// TIA Portal V16 export
// export: Created 2023-03-29T11:04:41.0167159Z, ExportSetting WithDefaults, DisplayName Totally Integrated Automation Portal, DisplayVersion V16 Update 6, DisplayName TIA Portal Version Control Interface, DisplayVersion V16 Update 2, DisplayName TIA Portal Openness, DisplayVersion V16 Update 6, DisplayName STEP 7 Professional, DisplayVersion V16 Update 6, DisplayName STEP 7 Safety, DisplayVersion V16, DisplayName WinCC Advanced, DisplayVersion V16 Update 6
FUNCTION "Synchroniczna_wymiana_danych_PLC1-PLC2" : Void   // FC61, LAD
TITLE = Wymiana danych
{ S7_Optimized_Access := 'TRUE' }
AUTHOR : rtecmer
VERSION : 0.1
// Funkcja grupuje bloki funkcji służąc wymianie danych HMI - PLC1, HMI-PLC2 i SCADA. Wprowadzanie wartości z poziomu HMI Zbiorniki lub HMI Pompownia czy SCADA jest nadpisywane w docelowym sterowniku. Zmian włónych parametrów układu sterowania pompownią, zbiornikami można dokonywać w dowolnego miejsca.
// stored: AutoNumber true, IsIECCheckEnabled false, SetENOAutomatically false, UDAEnableTagReadback false
   VAR_TEMP   // added for the SCL form of the ladder/FBD networks
      _w1 : Bool;
   END_VAR
BEGIN

REGION Network 2: Detekcja zmiany danych - Poziom napełnienia
   // Wymiana danych między PLC 1, PLC 2, SCADA
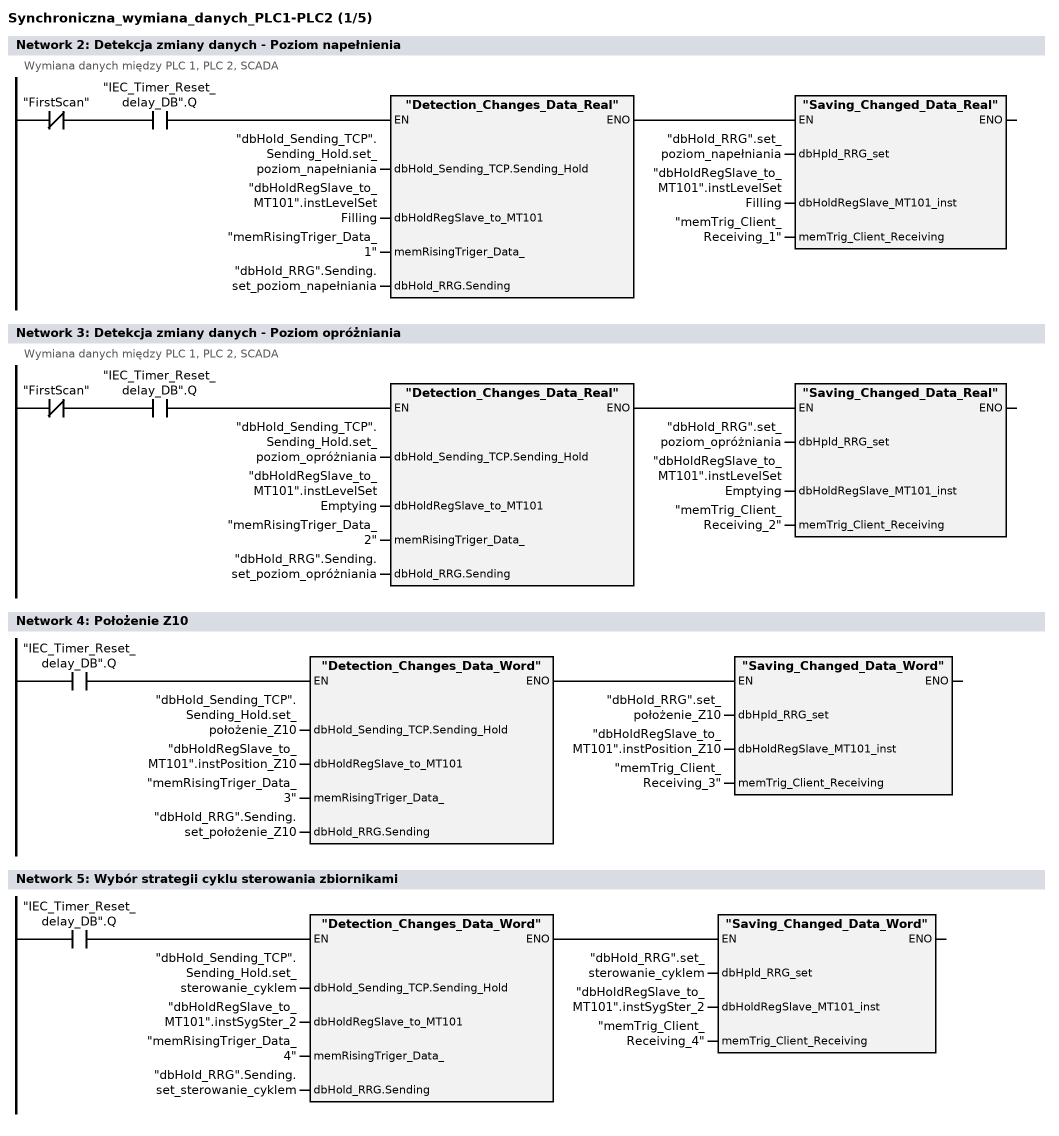
   RUNG wire#powerrail
      I_Contact( "FirstScan" )
      Contact( "IEC_Timer_Reset_delay_DB".Q )
      "Detection_Changes_Data_Real"("dbHold_Sending_TCP.Sending_Hold" := "dbHold_Sending_TCP".Sending_Hold.set_poziom_napełniania, dbHoldRegSlave_to_MT101 := "dbHoldRegSlave_to_MT101".instLevelSetFilling, memRisingTriger_Data_ := "memRisingTriger_Data_1", "dbHold_RRG.Sending" := "dbHold_RRG".Sending.set_poziom_napełniania)
      "Saving_Changed_Data_Real"(dbHpld_RRG_set := "dbHold_RRG".set_poziom_napełniania, dbHoldRegSlave_MT101_inst := "dbHoldRegSlave_to_MT101".instLevelSetFilling, memTrig_Client_Receiving := "memTrig_Client_Receiving_1")
   END_RUNG
   // the same network as SCL:
   "Detection_Changes_Data_Real"(EN := NOT "FirstScan" AND "IEC_Timer_Reset_delay_DB".Q,
                           "dbHold_Sending_TCP.Sending_Hold" := "dbHold_Sending_TCP".Sending_Hold.set_poziom_napełniania,
                           dbHoldRegSlave_to_MT101 := "dbHoldRegSlave_to_MT101".instLevelSetFilling,
                           memRisingTriger_Data_ := "memRisingTriger_Data_1",
                           "dbHold_RRG.Sending" := "dbHold_RRG".Sending.set_poziom_napełniania,
                           ENO => #_w1);
   IF #_w1 THEN
       "Saving_Changed_Data_Real"(dbHpld_RRG_set := "dbHold_RRG".set_poziom_napełniania,
                               dbHoldRegSlave_MT101_inst := "dbHoldRegSlave_to_MT101".instLevelSetFilling,
                               memTrig_Client_Receiving := "memTrig_Client_Receiving_1");
   END_IF;
END_REGION

REGION Network 3: Detekcja zmiany danych - Poziom opróżniania
   // Wymiana danych między PLC 1, PLC 2, SCADA
   RUNG wire#powerrail
      I_Contact( "FirstScan" )
      Contact( "IEC_Timer_Reset_delay_DB".Q )
      "Detection_Changes_Data_Real"("dbHold_Sending_TCP.Sending_Hold" := "dbHold_Sending_TCP".Sending_Hold.set_poziom_opróżniania, dbHoldRegSlave_to_MT101 := "dbHoldRegSlave_to_MT101".instLevelSetEmptying, memRisingTriger_Data_ := "memRisingTriger_Data_2", "dbHold_RRG.Sending" := "dbHold_RRG".Sending.set_poziom_opróżniania)
      "Saving_Changed_Data_Real"(dbHpld_RRG_set := "dbHold_RRG".set_poziom_opróżniania, dbHoldRegSlave_MT101_inst := "dbHoldRegSlave_to_MT101".instLevelSetEmptying, memTrig_Client_Receiving := "memTrig_Client_Receiving_2")
   END_RUNG
   // the same network as SCL:
   "Detection_Changes_Data_Real"(EN := NOT "FirstScan" AND "IEC_Timer_Reset_delay_DB".Q,
                           "dbHold_Sending_TCP.Sending_Hold" := "dbHold_Sending_TCP".Sending_Hold.set_poziom_opróżniania,
                           dbHoldRegSlave_to_MT101 := "dbHoldRegSlave_to_MT101".instLevelSetEmptying,
                           memRisingTriger_Data_ := "memRisingTriger_Data_2",
                           "dbHold_RRG.Sending" := "dbHold_RRG".Sending.set_poziom_opróżniania,
                           ENO => #_w1);
   IF #_w1 THEN
       "Saving_Changed_Data_Real"(dbHpld_RRG_set := "dbHold_RRG".set_poziom_opróżniania,
                               dbHoldRegSlave_MT101_inst := "dbHoldRegSlave_to_MT101".instLevelSetEmptying,
                               memTrig_Client_Receiving := "memTrig_Client_Receiving_2");
   END_IF;
END_REGION

REGION Network 4: Położenie Z10
   RUNG wire#powerrail
      Contact( "IEC_Timer_Reset_delay_DB".Q )
      "Detection_Changes_Data_Word"("dbHold_Sending_TCP.Sending_Hold" := "dbHold_Sending_TCP".Sending_Hold.set_położenie_Z10, dbHoldRegSlave_to_MT101 := "dbHoldRegSlave_to_MT101".instPosition_Z10, memRisingTriger_Data_ := "memRisingTriger_Data_3", "dbHold_RRG.Sending" := "dbHold_RRG".Sending.set_położenie_Z10)
      "Saving_Changed_Data_Word"(dbHpld_RRG_set := "dbHold_RRG".set_położenie_Z10, dbHoldRegSlave_MT101_inst := "dbHoldRegSlave_to_MT101".instPosition_Z10, memTrig_Client_Receiving := "memTrig_Client_Receiving_3")
   END_RUNG
   // the same network as SCL:
   "Detection_Changes_Data_Word"(EN := "IEC_Timer_Reset_delay_DB".Q,
                           "dbHold_Sending_TCP.Sending_Hold" := "dbHold_Sending_TCP".Sending_Hold.set_położenie_Z10,
                           dbHoldRegSlave_to_MT101 := "dbHoldRegSlave_to_MT101".instPosition_Z10,
                           memRisingTriger_Data_ := "memRisingTriger_Data_3",
                           "dbHold_RRG.Sending" := "dbHold_RRG".Sending.set_położenie_Z10,
                           ENO => #_w1);
   IF #_w1 THEN
       "Saving_Changed_Data_Word"(dbHpld_RRG_set := "dbHold_RRG".set_położenie_Z10,
                               dbHoldRegSlave_MT101_inst := "dbHoldRegSlave_to_MT101".instPosition_Z10,
                               memTrig_Client_Receiving := "memTrig_Client_Receiving_3");
   END_IF;
END_REGION

REGION Network 5: Wybór strategii cyklu sterowania zbiornikami
   RUNG wire#powerrail
      Contact( "IEC_Timer_Reset_delay_DB".Q )
      "Detection_Changes_Data_Word"("dbHold_Sending_TCP.Sending_Hold" := "dbHold_Sending_TCP".Sending_Hold.set_sterowanie_cyklem, dbHoldRegSlave_to_MT101 := "dbHoldRegSlave_to_MT101".instSygSter_2, memRisingTriger_Data_ := "memRisingTriger_Data_4", "dbHold_RRG.Sending" := "dbHold_RRG".Sending.set_sterowanie_cyklem)
      "Saving_Changed_Data_Word"(dbHpld_RRG_set := "dbHold_RRG".set_sterowanie_cyklem, dbHoldRegSlave_MT101_inst := "dbHoldRegSlave_to_MT101".instSygSter_2, memTrig_Client_Receiving := "memTrig_Client_Receiving_4")
   END_RUNG
   // the same network as SCL:
   "Detection_Changes_Data_Word"(EN := "IEC_Timer_Reset_delay_DB".Q,
                           "dbHold_Sending_TCP.Sending_Hold" := "dbHold_Sending_TCP".Sending_Hold.set_sterowanie_cyklem,
                           dbHoldRegSlave_to_MT101 := "dbHoldRegSlave_to_MT101".instSygSter_2,
                           memRisingTriger_Data_ := "memRisingTriger_Data_4",
                           "dbHold_RRG.Sending" := "dbHold_RRG".Sending.set_sterowanie_cyklem,
                           ENO => #_w1);
   IF #_w1 THEN
       "Saving_Changed_Data_Word"(dbHpld_RRG_set := "dbHold_RRG".set_sterowanie_cyklem,
                               dbHoldRegSlave_MT101_inst := "dbHoldRegSlave_to_MT101".instSygSter_2,
                               memTrig_Client_Receiving := "memTrig_Client_Receiving_4");
   END_IF;
END_REGION

REGION Network 6: Godzina napełniania start
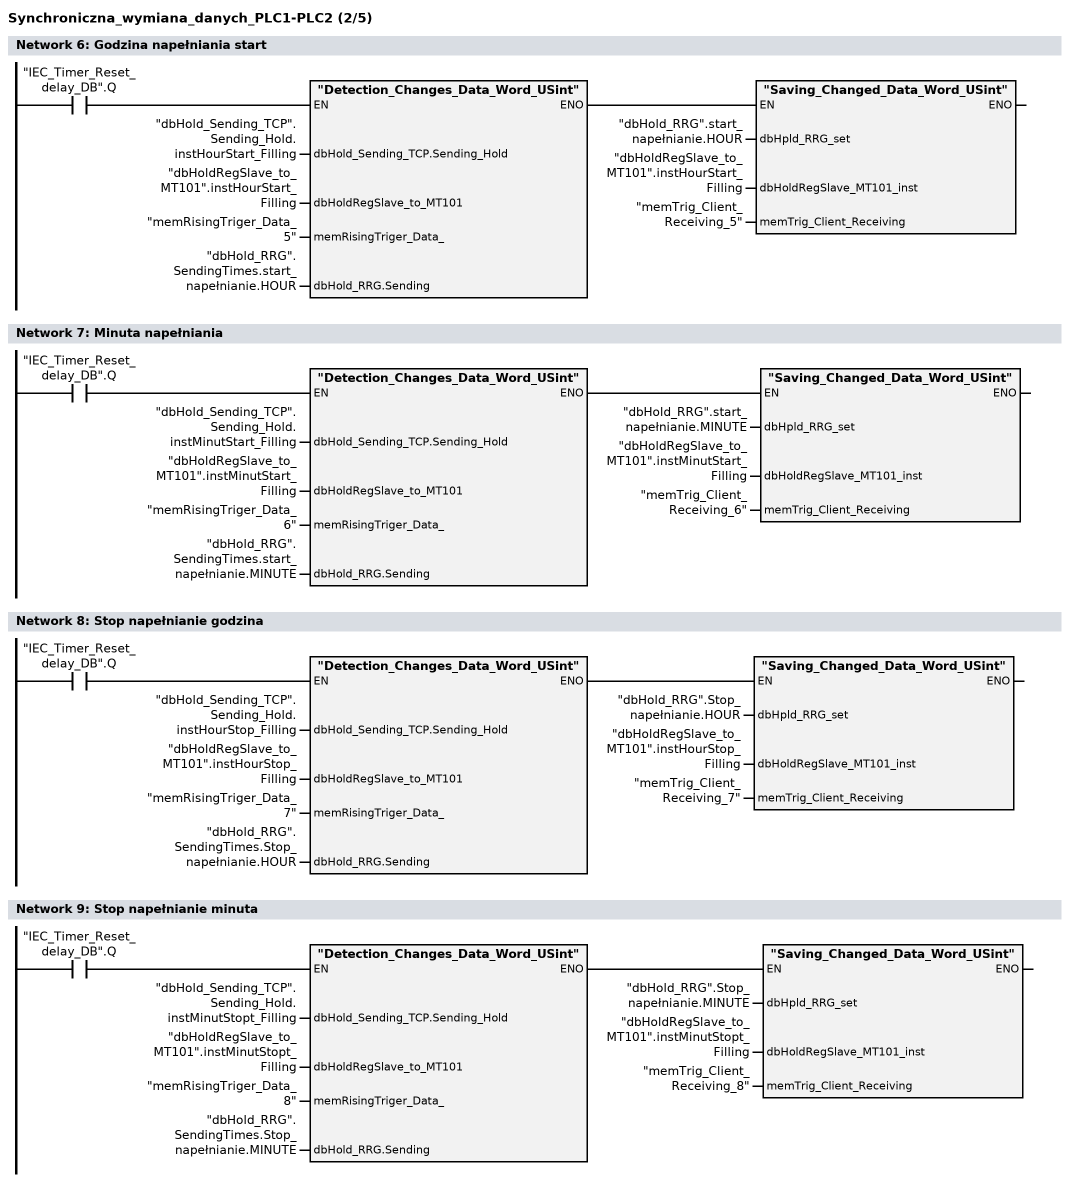
   RUNG wire#powerrail
      Contact( "IEC_Timer_Reset_delay_DB".Q )
      "Detection_Changes_Data_Word_USint"("dbHold_Sending_TCP.Sending_Hold" := "dbHold_Sending_TCP".Sending_Hold.instHourStart_Filling, dbHoldRegSlave_to_MT101 := "dbHoldRegSlave_to_MT101".instHourStart_Filling, memRisingTriger_Data_ := "memRisingTriger_Data_5", "dbHold_RRG.Sending" := "dbHold_RRG".SendingTimes.start_napełnianie.HOUR)
      "Saving_Changed_Data_Word_USint"(dbHpld_RRG_set := "dbHold_RRG".start_napełnianie.HOUR, dbHoldRegSlave_MT101_inst := "dbHoldRegSlave_to_MT101".instHourStart_Filling, memTrig_Client_Receiving := "memTrig_Client_Receiving_5")
   END_RUNG
   // the same network as SCL:
   "Detection_Changes_Data_Word_USint"(EN := "IEC_Timer_Reset_delay_DB".Q,
                           "dbHold_Sending_TCP.Sending_Hold" := "dbHold_Sending_TCP".Sending_Hold.instHourStart_Filling,
                           dbHoldRegSlave_to_MT101 := "dbHoldRegSlave_to_MT101".instHourStart_Filling,
                           memRisingTriger_Data_ := "memRisingTriger_Data_5",
                           "dbHold_RRG.Sending" := "dbHold_RRG".SendingTimes.start_napełnianie.HOUR,
                           ENO => #_w1);
   IF #_w1 THEN
       "Saving_Changed_Data_Word_USint"(dbHpld_RRG_set := "dbHold_RRG".start_napełnianie.HOUR,
                               dbHoldRegSlave_MT101_inst := "dbHoldRegSlave_to_MT101".instHourStart_Filling,
                               memTrig_Client_Receiving := "memTrig_Client_Receiving_5");
   END_IF;
END_REGION

REGION Network 7: Minuta napełniania
   RUNG wire#powerrail
      Contact( "IEC_Timer_Reset_delay_DB".Q )
      "Detection_Changes_Data_Word_USint"("dbHold_Sending_TCP.Sending_Hold" := "dbHold_Sending_TCP".Sending_Hold.instMinutStart_Filling, dbHoldRegSlave_to_MT101 := "dbHoldRegSlave_to_MT101".instMinutStart_Filling, memRisingTriger_Data_ := "memRisingTriger_Data_6", "dbHold_RRG.Sending" := "dbHold_RRG".SendingTimes.start_napełnianie.MINUTE)
      "Saving_Changed_Data_Word_USint"(dbHpld_RRG_set := "dbHold_RRG".start_napełnianie.MINUTE, dbHoldRegSlave_MT101_inst := "dbHoldRegSlave_to_MT101".instMinutStart_Filling, memTrig_Client_Receiving := "memTrig_Client_Receiving_6")
   END_RUNG
   // the same network as SCL:
   "Detection_Changes_Data_Word_USint"(EN := "IEC_Timer_Reset_delay_DB".Q,
                           "dbHold_Sending_TCP.Sending_Hold" := "dbHold_Sending_TCP".Sending_Hold.instMinutStart_Filling,
                           dbHoldRegSlave_to_MT101 := "dbHoldRegSlave_to_MT101".instMinutStart_Filling,
                           memRisingTriger_Data_ := "memRisingTriger_Data_6",
                           "dbHold_RRG.Sending" := "dbHold_RRG".SendingTimes.start_napełnianie.MINUTE,
                           ENO => #_w1);
   IF #_w1 THEN
       "Saving_Changed_Data_Word_USint"(dbHpld_RRG_set := "dbHold_RRG".start_napełnianie.MINUTE,
                               dbHoldRegSlave_MT101_inst := "dbHoldRegSlave_to_MT101".instMinutStart_Filling,
                               memTrig_Client_Receiving := "memTrig_Client_Receiving_6");
   END_IF;
END_REGION

REGION Network 8: Stop napełnianie godzina
   RUNG wire#powerrail
      Contact( "IEC_Timer_Reset_delay_DB".Q )
      "Detection_Changes_Data_Word_USint"("dbHold_Sending_TCP.Sending_Hold" := "dbHold_Sending_TCP".Sending_Hold.instHourStop_Filling, dbHoldRegSlave_to_MT101 := "dbHoldRegSlave_to_MT101".instHourStop_Filling, memRisingTriger_Data_ := "memRisingTriger_Data_7", "dbHold_RRG.Sending" := "dbHold_RRG".SendingTimes.Stop_napełnianie.HOUR)
      "Saving_Changed_Data_Word_USint"(dbHpld_RRG_set := "dbHold_RRG".Stop_napełnianie.HOUR, dbHoldRegSlave_MT101_inst := "dbHoldRegSlave_to_MT101".instHourStop_Filling, memTrig_Client_Receiving := "memTrig_Client_Receiving_7")
   END_RUNG
   // the same network as SCL:
   "Detection_Changes_Data_Word_USint"(EN := "IEC_Timer_Reset_delay_DB".Q,
                           "dbHold_Sending_TCP.Sending_Hold" := "dbHold_Sending_TCP".Sending_Hold.instHourStop_Filling,
                           dbHoldRegSlave_to_MT101 := "dbHoldRegSlave_to_MT101".instHourStop_Filling,
                           memRisingTriger_Data_ := "memRisingTriger_Data_7",
                           "dbHold_RRG.Sending" := "dbHold_RRG".SendingTimes.Stop_napełnianie.HOUR,
                           ENO => #_w1);
   IF #_w1 THEN
       "Saving_Changed_Data_Word_USint"(dbHpld_RRG_set := "dbHold_RRG".Stop_napełnianie.HOUR,
                               dbHoldRegSlave_MT101_inst := "dbHoldRegSlave_to_MT101".instHourStop_Filling,
                               memTrig_Client_Receiving := "memTrig_Client_Receiving_7");
   END_IF;
END_REGION

REGION Network 9: Stop napełnianie minuta
   RUNG wire#powerrail
      Contact( "IEC_Timer_Reset_delay_DB".Q )
      "Detection_Changes_Data_Word_USint"("dbHold_Sending_TCP.Sending_Hold" := "dbHold_Sending_TCP".Sending_Hold.instMinutStopt_Filling, dbHoldRegSlave_to_MT101 := "dbHoldRegSlave_to_MT101".instMinutStopt_Filling, memRisingTriger_Data_ := "memRisingTriger_Data_8", "dbHold_RRG.Sending" := "dbHold_RRG".SendingTimes.Stop_napełnianie.MINUTE)
      "Saving_Changed_Data_Word_USint"(dbHpld_RRG_set := "dbHold_RRG".Stop_napełnianie.MINUTE, dbHoldRegSlave_MT101_inst := "dbHoldRegSlave_to_MT101".instMinutStopt_Filling, memTrig_Client_Receiving := "memTrig_Client_Receiving_8")
   END_RUNG
   // the same network as SCL:
   "Detection_Changes_Data_Word_USint"(EN := "IEC_Timer_Reset_delay_DB".Q,
                           "dbHold_Sending_TCP.Sending_Hold" := "dbHold_Sending_TCP".Sending_Hold.instMinutStopt_Filling,
                           dbHoldRegSlave_to_MT101 := "dbHoldRegSlave_to_MT101".instMinutStopt_Filling,
                           memRisingTriger_Data_ := "memRisingTriger_Data_8",
                           "dbHold_RRG.Sending" := "dbHold_RRG".SendingTimes.Stop_napełnianie.MINUTE,
                           ENO => #_w1);
   IF #_w1 THEN
       "Saving_Changed_Data_Word_USint"(dbHpld_RRG_set := "dbHold_RRG".Stop_napełnianie.MINUTE,
                               dbHoldRegSlave_MT101_inst := "dbHoldRegSlave_to_MT101".instMinutStopt_Filling,
                               memTrig_Client_Receiving := "memTrig_Client_Receiving_8");
   END_IF;
END_REGION

REGION Network 10: Start przetłaczanie (miasto) godzina
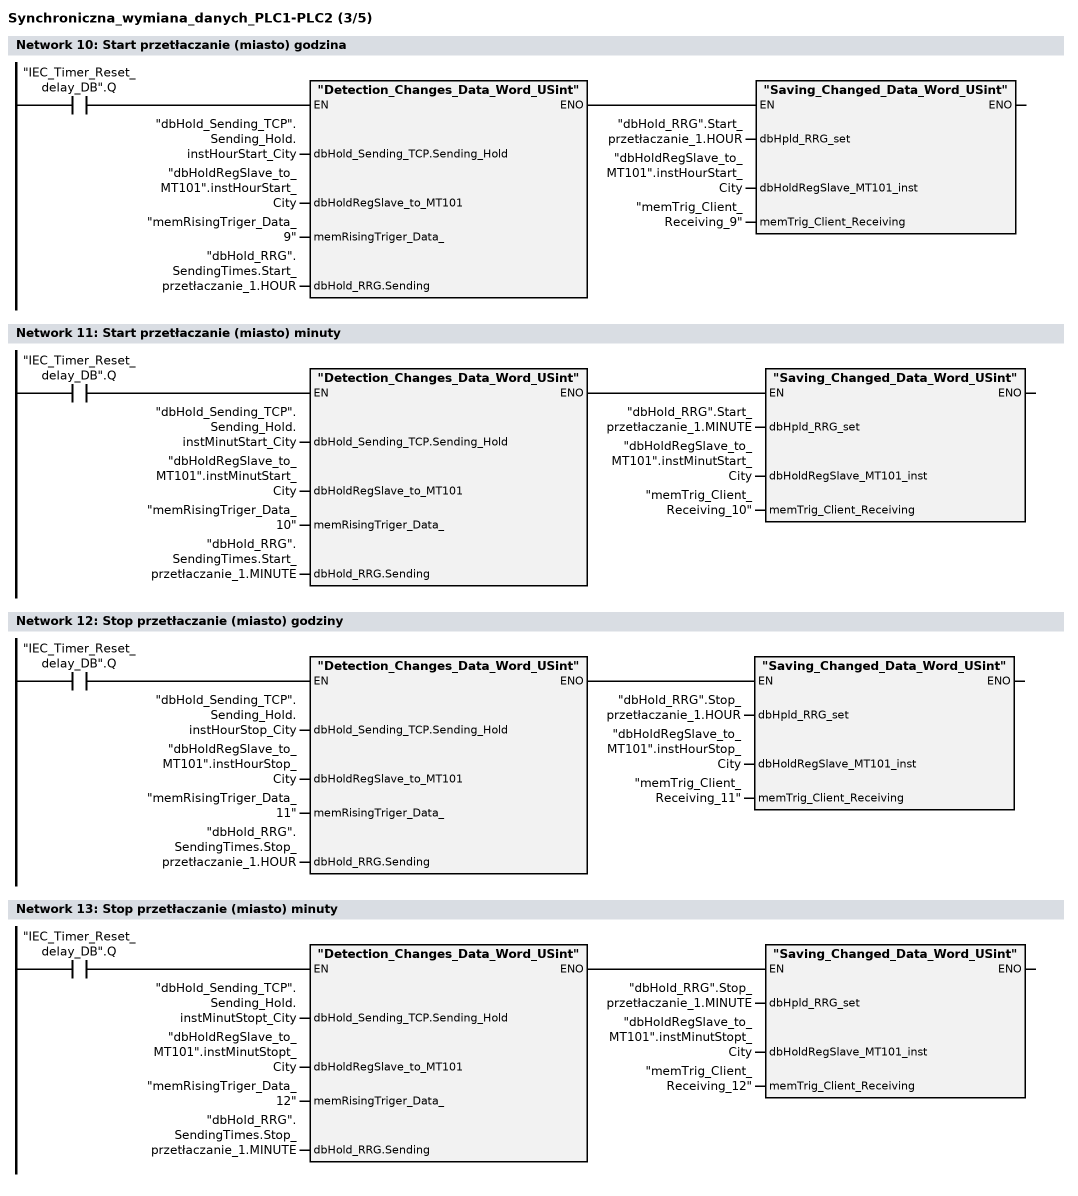
   RUNG wire#powerrail
      Contact( "IEC_Timer_Reset_delay_DB".Q )
      "Detection_Changes_Data_Word_USint"("dbHold_Sending_TCP.Sending_Hold" := "dbHold_Sending_TCP".Sending_Hold.instHourStart_City, dbHoldRegSlave_to_MT101 := "dbHoldRegSlave_to_MT101".instHourStart_City, memRisingTriger_Data_ := "memRisingTriger_Data_9", "dbHold_RRG.Sending" := "dbHold_RRG".SendingTimes.Start_przetłaczanie_1.HOUR)
      "Saving_Changed_Data_Word_USint"(dbHpld_RRG_set := "dbHold_RRG".Start_przetłaczanie_1.HOUR, dbHoldRegSlave_MT101_inst := "dbHoldRegSlave_to_MT101".instHourStart_City, memTrig_Client_Receiving := "memTrig_Client_Receiving_9")
   END_RUNG
   // the same network as SCL:
   "Detection_Changes_Data_Word_USint"(EN := "IEC_Timer_Reset_delay_DB".Q,
                           "dbHold_Sending_TCP.Sending_Hold" := "dbHold_Sending_TCP".Sending_Hold.instHourStart_City,
                           dbHoldRegSlave_to_MT101 := "dbHoldRegSlave_to_MT101".instHourStart_City,
                           memRisingTriger_Data_ := "memRisingTriger_Data_9",
                           "dbHold_RRG.Sending" := "dbHold_RRG".SendingTimes.Start_przetłaczanie_1.HOUR,
                           ENO => #_w1);
   IF #_w1 THEN
       "Saving_Changed_Data_Word_USint"(dbHpld_RRG_set := "dbHold_RRG".Start_przetłaczanie_1.HOUR,
                               dbHoldRegSlave_MT101_inst := "dbHoldRegSlave_to_MT101".instHourStart_City,
                               memTrig_Client_Receiving := "memTrig_Client_Receiving_9");
   END_IF;
END_REGION

REGION Network 11: Start przetłaczanie (miasto) minuty
   RUNG wire#powerrail
      Contact( "IEC_Timer_Reset_delay_DB".Q )
      "Detection_Changes_Data_Word_USint"("dbHold_Sending_TCP.Sending_Hold" := "dbHold_Sending_TCP".Sending_Hold.instMinutStart_City, dbHoldRegSlave_to_MT101 := "dbHoldRegSlave_to_MT101".instMinutStart_City, memRisingTriger_Data_ := "memRisingTriger_Data_10", "dbHold_RRG.Sending" := "dbHold_RRG".SendingTimes.Start_przetłaczanie_1.MINUTE)
      "Saving_Changed_Data_Word_USint"(dbHpld_RRG_set := "dbHold_RRG".Start_przetłaczanie_1.MINUTE, dbHoldRegSlave_MT101_inst := "dbHoldRegSlave_to_MT101".instMinutStart_City, memTrig_Client_Receiving := "memTrig_Client_Receiving_10")
   END_RUNG
   // the same network as SCL:
   "Detection_Changes_Data_Word_USint"(EN := "IEC_Timer_Reset_delay_DB".Q,
                           "dbHold_Sending_TCP.Sending_Hold" := "dbHold_Sending_TCP".Sending_Hold.instMinutStart_City,
                           dbHoldRegSlave_to_MT101 := "dbHoldRegSlave_to_MT101".instMinutStart_City,
                           memRisingTriger_Data_ := "memRisingTriger_Data_10",
                           "dbHold_RRG.Sending" := "dbHold_RRG".SendingTimes.Start_przetłaczanie_1.MINUTE,
                           ENO => #_w1);
   IF #_w1 THEN
       "Saving_Changed_Data_Word_USint"(dbHpld_RRG_set := "dbHold_RRG".Start_przetłaczanie_1.MINUTE,
                               dbHoldRegSlave_MT101_inst := "dbHoldRegSlave_to_MT101".instMinutStart_City,
                               memTrig_Client_Receiving := "memTrig_Client_Receiving_10");
   END_IF;
END_REGION

REGION Network 12: Stop przetłaczanie (miasto) godziny
   RUNG wire#powerrail
      Contact( "IEC_Timer_Reset_delay_DB".Q )
      "Detection_Changes_Data_Word_USint"("dbHold_Sending_TCP.Sending_Hold" := "dbHold_Sending_TCP".Sending_Hold.instHourStop_City, dbHoldRegSlave_to_MT101 := "dbHoldRegSlave_to_MT101".instHourStop_City, memRisingTriger_Data_ := "memRisingTriger_Data_11", "dbHold_RRG.Sending" := "dbHold_RRG".SendingTimes.Stop_przetłaczanie_1.HOUR)
      "Saving_Changed_Data_Word_USint"(dbHpld_RRG_set := "dbHold_RRG".Stop_przetłaczanie_1.HOUR, dbHoldRegSlave_MT101_inst := "dbHoldRegSlave_to_MT101".instHourStop_City, memTrig_Client_Receiving := "memTrig_Client_Receiving_11")
   END_RUNG
   // the same network as SCL:
   "Detection_Changes_Data_Word_USint"(EN := "IEC_Timer_Reset_delay_DB".Q,
                           "dbHold_Sending_TCP.Sending_Hold" := "dbHold_Sending_TCP".Sending_Hold.instHourStop_City,
                           dbHoldRegSlave_to_MT101 := "dbHoldRegSlave_to_MT101".instHourStop_City,
                           memRisingTriger_Data_ := "memRisingTriger_Data_11",
                           "dbHold_RRG.Sending" := "dbHold_RRG".SendingTimes.Stop_przetłaczanie_1.HOUR,
                           ENO => #_w1);
   IF #_w1 THEN
       "Saving_Changed_Data_Word_USint"(dbHpld_RRG_set := "dbHold_RRG".Stop_przetłaczanie_1.HOUR,
                               dbHoldRegSlave_MT101_inst := "dbHoldRegSlave_to_MT101".instHourStop_City,
                               memTrig_Client_Receiving := "memTrig_Client_Receiving_11");
   END_IF;
END_REGION

REGION Network 13: Stop przetłaczanie (miasto) minuty
   RUNG wire#powerrail
      Contact( "IEC_Timer_Reset_delay_DB".Q )
      "Detection_Changes_Data_Word_USint"("dbHold_Sending_TCP.Sending_Hold" := "dbHold_Sending_TCP".Sending_Hold.instMinutStopt_City, dbHoldRegSlave_to_MT101 := "dbHoldRegSlave_to_MT101".instMinutStopt_City, memRisingTriger_Data_ := "memRisingTriger_Data_12", "dbHold_RRG.Sending" := "dbHold_RRG".SendingTimes.Stop_przetłaczanie_1.MINUTE)
      "Saving_Changed_Data_Word_USint"(dbHpld_RRG_set := "dbHold_RRG".Stop_przetłaczanie_1.MINUTE, dbHoldRegSlave_MT101_inst := "dbHoldRegSlave_to_MT101".instMinutStopt_City, memTrig_Client_Receiving := "memTrig_Client_Receiving_12")
   END_RUNG
   // the same network as SCL:
   "Detection_Changes_Data_Word_USint"(EN := "IEC_Timer_Reset_delay_DB".Q,
                           "dbHold_Sending_TCP.Sending_Hold" := "dbHold_Sending_TCP".Sending_Hold.instMinutStopt_City,
                           dbHoldRegSlave_to_MT101 := "dbHoldRegSlave_to_MT101".instMinutStopt_City,
                           memRisingTriger_Data_ := "memRisingTriger_Data_12",
                           "dbHold_RRG.Sending" := "dbHold_RRG".SendingTimes.Stop_przetłaczanie_1.MINUTE,
                           ENO => #_w1);
   IF #_w1 THEN
       "Saving_Changed_Data_Word_USint"(dbHpld_RRG_set := "dbHold_RRG".Stop_przetłaczanie_1.MINUTE,
                               dbHoldRegSlave_MT101_inst := "dbHoldRegSlave_to_MT101".instMinutStopt_City,
                               memTrig_Client_Receiving := "memTrig_Client_Receiving_12");
   END_IF;
END_REGION

REGION Network 14: Start dosilanie godziny
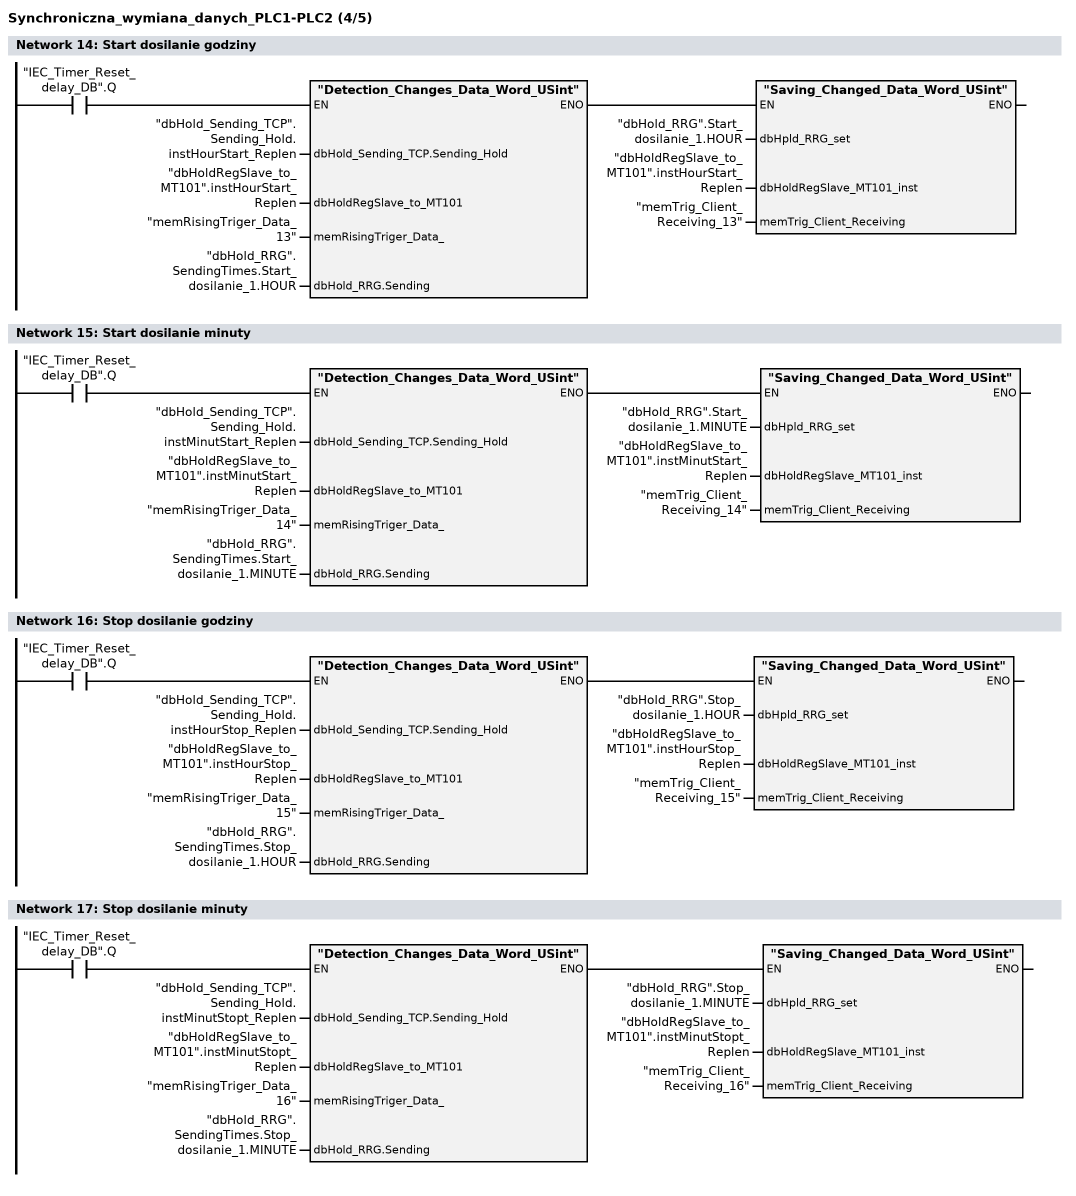
   RUNG wire#powerrail
      Contact( "IEC_Timer_Reset_delay_DB".Q )
      "Detection_Changes_Data_Word_USint"("dbHold_Sending_TCP.Sending_Hold" := "dbHold_Sending_TCP".Sending_Hold.instHourStart_Replen, dbHoldRegSlave_to_MT101 := "dbHoldRegSlave_to_MT101".instHourStart_Replen, memRisingTriger_Data_ := "memRisingTriger_Data_13", "dbHold_RRG.Sending" := "dbHold_RRG".SendingTimes.Start_dosilanie_1.HOUR)
      "Saving_Changed_Data_Word_USint"(dbHpld_RRG_set := "dbHold_RRG".Start_dosilanie_1.HOUR, dbHoldRegSlave_MT101_inst := "dbHoldRegSlave_to_MT101".instHourStart_Replen, memTrig_Client_Receiving := "memTrig_Client_Receiving_13")
   END_RUNG
   // the same network as SCL:
   "Detection_Changes_Data_Word_USint"(EN := "IEC_Timer_Reset_delay_DB".Q,
                           "dbHold_Sending_TCP.Sending_Hold" := "dbHold_Sending_TCP".Sending_Hold.instHourStart_Replen,
                           dbHoldRegSlave_to_MT101 := "dbHoldRegSlave_to_MT101".instHourStart_Replen,
                           memRisingTriger_Data_ := "memRisingTriger_Data_13",
                           "dbHold_RRG.Sending" := "dbHold_RRG".SendingTimes.Start_dosilanie_1.HOUR,
                           ENO => #_w1);
   IF #_w1 THEN
       "Saving_Changed_Data_Word_USint"(dbHpld_RRG_set := "dbHold_RRG".Start_dosilanie_1.HOUR,
                               dbHoldRegSlave_MT101_inst := "dbHoldRegSlave_to_MT101".instHourStart_Replen,
                               memTrig_Client_Receiving := "memTrig_Client_Receiving_13");
   END_IF;
END_REGION

REGION Network 15: Start dosilanie minuty
   RUNG wire#powerrail
      Contact( "IEC_Timer_Reset_delay_DB".Q )
      "Detection_Changes_Data_Word_USint"("dbHold_Sending_TCP.Sending_Hold" := "dbHold_Sending_TCP".Sending_Hold.instMinutStart_Replen, dbHoldRegSlave_to_MT101 := "dbHoldRegSlave_to_MT101".instMinutStart_Replen, memRisingTriger_Data_ := "memRisingTriger_Data_14", "dbHold_RRG.Sending" := "dbHold_RRG".SendingTimes.Start_dosilanie_1.MINUTE)
      "Saving_Changed_Data_Word_USint"(dbHpld_RRG_set := "dbHold_RRG".Start_dosilanie_1.MINUTE, dbHoldRegSlave_MT101_inst := "dbHoldRegSlave_to_MT101".instMinutStart_Replen, memTrig_Client_Receiving := "memTrig_Client_Receiving_14")
   END_RUNG
   // the same network as SCL:
   "Detection_Changes_Data_Word_USint"(EN := "IEC_Timer_Reset_delay_DB".Q,
                           "dbHold_Sending_TCP.Sending_Hold" := "dbHold_Sending_TCP".Sending_Hold.instMinutStart_Replen,
                           dbHoldRegSlave_to_MT101 := "dbHoldRegSlave_to_MT101".instMinutStart_Replen,
                           memRisingTriger_Data_ := "memRisingTriger_Data_14",
                           "dbHold_RRG.Sending" := "dbHold_RRG".SendingTimes.Start_dosilanie_1.MINUTE,
                           ENO => #_w1);
   IF #_w1 THEN
       "Saving_Changed_Data_Word_USint"(dbHpld_RRG_set := "dbHold_RRG".Start_dosilanie_1.MINUTE,
                               dbHoldRegSlave_MT101_inst := "dbHoldRegSlave_to_MT101".instMinutStart_Replen,
                               memTrig_Client_Receiving := "memTrig_Client_Receiving_14");
   END_IF;
END_REGION

REGION Network 16: Stop dosilanie godziny
   RUNG wire#powerrail
      Contact( "IEC_Timer_Reset_delay_DB".Q )
      "Detection_Changes_Data_Word_USint"("dbHold_Sending_TCP.Sending_Hold" := "dbHold_Sending_TCP".Sending_Hold.instHourStop_Replen, dbHoldRegSlave_to_MT101 := "dbHoldRegSlave_to_MT101".instHourStop_Replen, memRisingTriger_Data_ := "memRisingTriger_Data_15", "dbHold_RRG.Sending" := "dbHold_RRG".SendingTimes.Stop_dosilanie_1.HOUR)
      "Saving_Changed_Data_Word_USint"(dbHpld_RRG_set := "dbHold_RRG".Stop_dosilanie_1.HOUR, dbHoldRegSlave_MT101_inst := "dbHoldRegSlave_to_MT101".instHourStop_Replen, memTrig_Client_Receiving := "memTrig_Client_Receiving_15")
   END_RUNG
   // the same network as SCL:
   "Detection_Changes_Data_Word_USint"(EN := "IEC_Timer_Reset_delay_DB".Q,
                           "dbHold_Sending_TCP.Sending_Hold" := "dbHold_Sending_TCP".Sending_Hold.instHourStop_Replen,
                           dbHoldRegSlave_to_MT101 := "dbHoldRegSlave_to_MT101".instHourStop_Replen,
                           memRisingTriger_Data_ := "memRisingTriger_Data_15",
                           "dbHold_RRG.Sending" := "dbHold_RRG".SendingTimes.Stop_dosilanie_1.HOUR,
                           ENO => #_w1);
   IF #_w1 THEN
       "Saving_Changed_Data_Word_USint"(dbHpld_RRG_set := "dbHold_RRG".Stop_dosilanie_1.HOUR,
                               dbHoldRegSlave_MT101_inst := "dbHoldRegSlave_to_MT101".instHourStop_Replen,
                               memTrig_Client_Receiving := "memTrig_Client_Receiving_15");
   END_IF;
END_REGION

REGION Network 17: Stop dosilanie minuty
   RUNG wire#powerrail
      Contact( "IEC_Timer_Reset_delay_DB".Q )
      "Detection_Changes_Data_Word_USint"("dbHold_Sending_TCP.Sending_Hold" := "dbHold_Sending_TCP".Sending_Hold.instMinutStopt_Replen, dbHoldRegSlave_to_MT101 := "dbHoldRegSlave_to_MT101".instMinutStopt_Replen, memRisingTriger_Data_ := "memRisingTriger_Data_16", "dbHold_RRG.Sending" := "dbHold_RRG".SendingTimes.Stop_dosilanie_1.MINUTE)
      "Saving_Changed_Data_Word_USint"(dbHpld_RRG_set := "dbHold_RRG".Stop_dosilanie_1.MINUTE, dbHoldRegSlave_MT101_inst := "dbHoldRegSlave_to_MT101".instMinutStopt_Replen, memTrig_Client_Receiving := "memTrig_Client_Receiving_16")
   END_RUNG
   // the same network as SCL:
   "Detection_Changes_Data_Word_USint"(EN := "IEC_Timer_Reset_delay_DB".Q,
                           "dbHold_Sending_TCP.Sending_Hold" := "dbHold_Sending_TCP".Sending_Hold.instMinutStopt_Replen,
                           dbHoldRegSlave_to_MT101 := "dbHoldRegSlave_to_MT101".instMinutStopt_Replen,
                           memRisingTriger_Data_ := "memRisingTriger_Data_16",
                           "dbHold_RRG.Sending" := "dbHold_RRG".SendingTimes.Stop_dosilanie_1.MINUTE,
                           ENO => #_w1);
   IF #_w1 THEN
       "Saving_Changed_Data_Word_USint"(dbHpld_RRG_set := "dbHold_RRG".Stop_dosilanie_1.MINUTE,
                               dbHoldRegSlave_MT101_inst := "dbHoldRegSlave_to_MT101".instMinutStopt_Replen,
                               memTrig_Client_Receiving := "memTrig_Client_Receiving_16");
   END_IF;
END_REGION

REGION Network 19: Wybór trymu pracy M1,M2,M3,M4, Z1-Z8
   // dbHoldRegSlave_MT101 - tu wartość zadajemy 
   // dbHoldSending_TCP.Sending_Hold - z tą wzmienną porównujemy 
   // dbHold_REG.Sending - tu wysyłamy
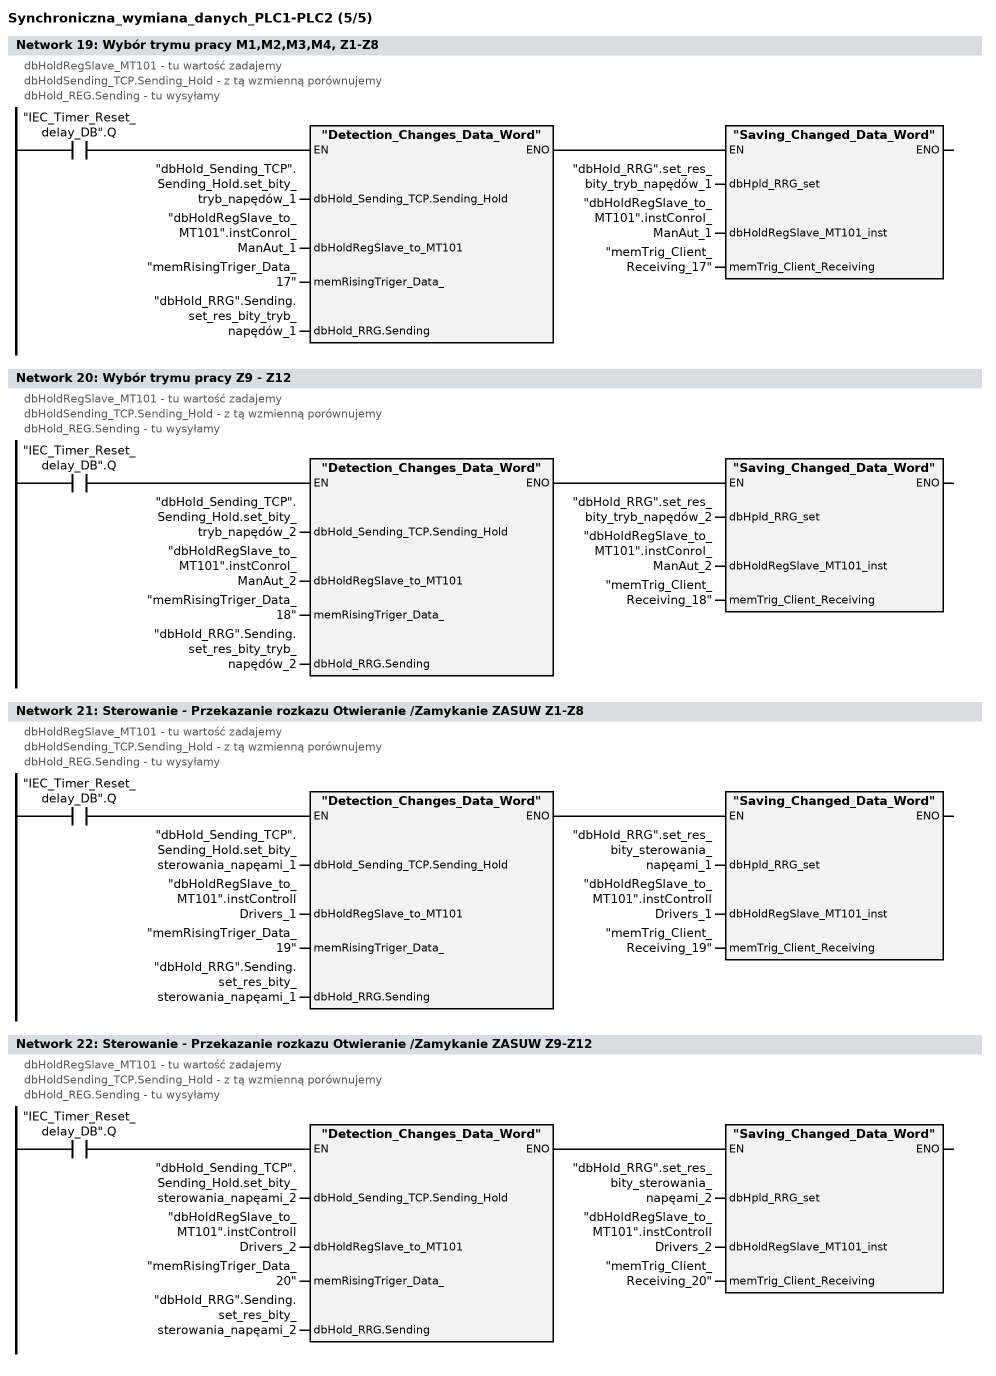
   RUNG wire#powerrail
      Contact( "IEC_Timer_Reset_delay_DB".Q )
      "Detection_Changes_Data_Word"("dbHold_Sending_TCP.Sending_Hold" := "dbHold_Sending_TCP".Sending_Hold.set_bity_tryb_napędów_1, dbHoldRegSlave_to_MT101 := "dbHoldRegSlave_to_MT101".instConrol_ManAut_1, memRisingTriger_Data_ := "memRisingTriger_Data_17", "dbHold_RRG.Sending" := "dbHold_RRG".Sending.set_res_bity_tryb_napędów_1)
      "Saving_Changed_Data_Word"(dbHpld_RRG_set := "dbHold_RRG".set_res_bity_tryb_napędów_1, dbHoldRegSlave_MT101_inst := "dbHoldRegSlave_to_MT101".instConrol_ManAut_1, memTrig_Client_Receiving := "memTrig_Client_Receiving_17")
   END_RUNG
   // the same network as SCL:
   "Detection_Changes_Data_Word"(EN := "IEC_Timer_Reset_delay_DB".Q,
                           "dbHold_Sending_TCP.Sending_Hold" := "dbHold_Sending_TCP".Sending_Hold.set_bity_tryb_napędów_1,
                           dbHoldRegSlave_to_MT101 := "dbHoldRegSlave_to_MT101".instConrol_ManAut_1,
                           memRisingTriger_Data_ := "memRisingTriger_Data_17",
                           "dbHold_RRG.Sending" := "dbHold_RRG".Sending.set_res_bity_tryb_napędów_1,
                           ENO => #_w1);
   IF #_w1 THEN
       "Saving_Changed_Data_Word"(dbHpld_RRG_set := "dbHold_RRG".set_res_bity_tryb_napędów_1,
                               dbHoldRegSlave_MT101_inst := "dbHoldRegSlave_to_MT101".instConrol_ManAut_1,
                               memTrig_Client_Receiving := "memTrig_Client_Receiving_17");
   END_IF;
END_REGION

REGION Network 20: Wybór trymu pracy Z9 - Z12
   // dbHoldRegSlave_MT101 - tu wartość zadajemy 
   // dbHoldSending_TCP.Sending_Hold - z tą wzmienną porównujemy 
   // dbHold_REG.Sending - tu wysyłamy
   RUNG wire#powerrail
      Contact( "IEC_Timer_Reset_delay_DB".Q )
      "Detection_Changes_Data_Word"("dbHold_Sending_TCP.Sending_Hold" := "dbHold_Sending_TCP".Sending_Hold.set_bity_tryb_napędów_2, dbHoldRegSlave_to_MT101 := "dbHoldRegSlave_to_MT101".instConrol_ManAut_2, memRisingTriger_Data_ := "memRisingTriger_Data_18", "dbHold_RRG.Sending" := "dbHold_RRG".Sending.set_res_bity_tryb_napędów_2)
      "Saving_Changed_Data_Word"(dbHpld_RRG_set := "dbHold_RRG".set_res_bity_tryb_napędów_2, dbHoldRegSlave_MT101_inst := "dbHoldRegSlave_to_MT101".instConrol_ManAut_2, memTrig_Client_Receiving := "memTrig_Client_Receiving_18")
   END_RUNG
   // the same network as SCL:
   "Detection_Changes_Data_Word"(EN := "IEC_Timer_Reset_delay_DB".Q,
                           "dbHold_Sending_TCP.Sending_Hold" := "dbHold_Sending_TCP".Sending_Hold.set_bity_tryb_napędów_2,
                           dbHoldRegSlave_to_MT101 := "dbHoldRegSlave_to_MT101".instConrol_ManAut_2,
                           memRisingTriger_Data_ := "memRisingTriger_Data_18",
                           "dbHold_RRG.Sending" := "dbHold_RRG".Sending.set_res_bity_tryb_napędów_2,
                           ENO => #_w1);
   IF #_w1 THEN
       "Saving_Changed_Data_Word"(dbHpld_RRG_set := "dbHold_RRG".set_res_bity_tryb_napędów_2,
                               dbHoldRegSlave_MT101_inst := "dbHoldRegSlave_to_MT101".instConrol_ManAut_2,
                               memTrig_Client_Receiving := "memTrig_Client_Receiving_18");
   END_IF;
END_REGION

REGION Network 21: Sterowanie - Przekazanie rozkazu Otwieranie /Zamykanie ZASUW Z1-Z8
   // dbHoldRegSlave_MT101 - tu wartość zadajemy 
   // dbHoldSending_TCP.Sending_Hold - z tą wzmienną porównujemy 
   // dbHold_REG.Sending - tu wysyłamy
   RUNG wire#powerrail
      Contact( "IEC_Timer_Reset_delay_DB".Q )
      "Detection_Changes_Data_Word"("dbHold_Sending_TCP.Sending_Hold" := "dbHold_Sending_TCP".Sending_Hold.set_bity_sterowania_napęami_1, dbHoldRegSlave_to_MT101 := "dbHoldRegSlave_to_MT101".instControllDrivers_1, memRisingTriger_Data_ := "memRisingTriger_Data_19", "dbHold_RRG.Sending" := "dbHold_RRG".Sending.set_res_bity_sterowania_napęami_1)
      "Saving_Changed_Data_Word"(dbHpld_RRG_set := "dbHold_RRG".set_res_bity_sterowania_napęami_1, dbHoldRegSlave_MT101_inst := "dbHoldRegSlave_to_MT101".instControllDrivers_1, memTrig_Client_Receiving := "memTrig_Client_Receiving_19")
   END_RUNG
   // the same network as SCL:
   "Detection_Changes_Data_Word"(EN := "IEC_Timer_Reset_delay_DB".Q,
                           "dbHold_Sending_TCP.Sending_Hold" := "dbHold_Sending_TCP".Sending_Hold.set_bity_sterowania_napęami_1,
                           dbHoldRegSlave_to_MT101 := "dbHoldRegSlave_to_MT101".instControllDrivers_1,
                           memRisingTriger_Data_ := "memRisingTriger_Data_19",
                           "dbHold_RRG.Sending" := "dbHold_RRG".Sending.set_res_bity_sterowania_napęami_1,
                           ENO => #_w1);
   IF #_w1 THEN
       "Saving_Changed_Data_Word"(dbHpld_RRG_set := "dbHold_RRG".set_res_bity_sterowania_napęami_1,
                               dbHoldRegSlave_MT101_inst := "dbHoldRegSlave_to_MT101".instControllDrivers_1,
                               memTrig_Client_Receiving := "memTrig_Client_Receiving_19");
   END_IF;
END_REGION

REGION Network 22: Sterowanie - Przekazanie rozkazu Otwieranie /Zamykanie ZASUW Z9-Z12
   // dbHoldRegSlave_MT101 - tu wartość zadajemy 
   // dbHoldSending_TCP.Sending_Hold - z tą wzmienną porównujemy 
   // dbHold_REG.Sending - tu wysyłamy
   RUNG wire#powerrail
      Contact( "IEC_Timer_Reset_delay_DB".Q )
      "Detection_Changes_Data_Word"("dbHold_Sending_TCP.Sending_Hold" := "dbHold_Sending_TCP".Sending_Hold.set_bity_sterowania_napęami_2, dbHoldRegSlave_to_MT101 := "dbHoldRegSlave_to_MT101".instControllDrivers_2, memRisingTriger_Data_ := "memRisingTriger_Data_20", "dbHold_RRG.Sending" := "dbHold_RRG".Sending.set_res_bity_sterowania_napęami_2)
      "Saving_Changed_Data_Word"(dbHpld_RRG_set := "dbHold_RRG".set_res_bity_sterowania_napęami_2, dbHoldRegSlave_MT101_inst := "dbHoldRegSlave_to_MT101".instControllDrivers_2, memTrig_Client_Receiving := "memTrig_Client_Receiving_20")
   END_RUNG
   // the same network as SCL:
   "Detection_Changes_Data_Word"(EN := "IEC_Timer_Reset_delay_DB".Q,
                           "dbHold_Sending_TCP.Sending_Hold" := "dbHold_Sending_TCP".Sending_Hold.set_bity_sterowania_napęami_2,
                           dbHoldRegSlave_to_MT101 := "dbHoldRegSlave_to_MT101".instControllDrivers_2,
                           memRisingTriger_Data_ := "memRisingTriger_Data_20",
                           "dbHold_RRG.Sending" := "dbHold_RRG".Sending.set_res_bity_sterowania_napęami_2,
                           ENO => #_w1);
   IF #_w1 THEN
       "Saving_Changed_Data_Word"(dbHpld_RRG_set := "dbHold_RRG".set_res_bity_sterowania_napęami_2,
                               dbHoldRegSlave_MT101_inst := "dbHoldRegSlave_to_MT101".instControllDrivers_2,
                               memTrig_Client_Receiving := "memTrig_Client_Receiving_20");
   END_IF;
END_REGION
END_FUNCTION
